(* PLC project TranslationStaging.project, CODESYS CODESYS V3.5 SP19 Patch 1 *)
(* stored: creationDateTime 2026-08-02T00:00:00, modificationDateTime 2026-08-02T00:00:00 *)

PROGRAM PRG_05_Translation_CFC
  VAR
    instTranslationArbiter : FB_TranslationArbiter;
    instSafetyTranslationM3 : FB_Safety_Translation;
    instTranslationRuntimeGate : FB_TranslationRuntimeGate;
    instTranslationM3 : FB_Translation;
    instTranslationFeedbackMemory : FB_TranslationFeedbackMemory;
    instTranslationRequestPublisher : FB_TranslationRequestPublisher;
    instTranslationCfcExpressions : FB_TranslationCfcExpressions;
  END_VAR
  VAR_OUTPUT
    TranslationFinalInterlockRequest : ST_TranslationFinalInterlockRequest;
    PowerCutOffRequested : BOOL;
    M3SafeStop : BOOL;
    M3PowerCutOff : BOOL;
    TranslationRequest : ST_TranslationFinalInterlockRequest;
  END_VAR

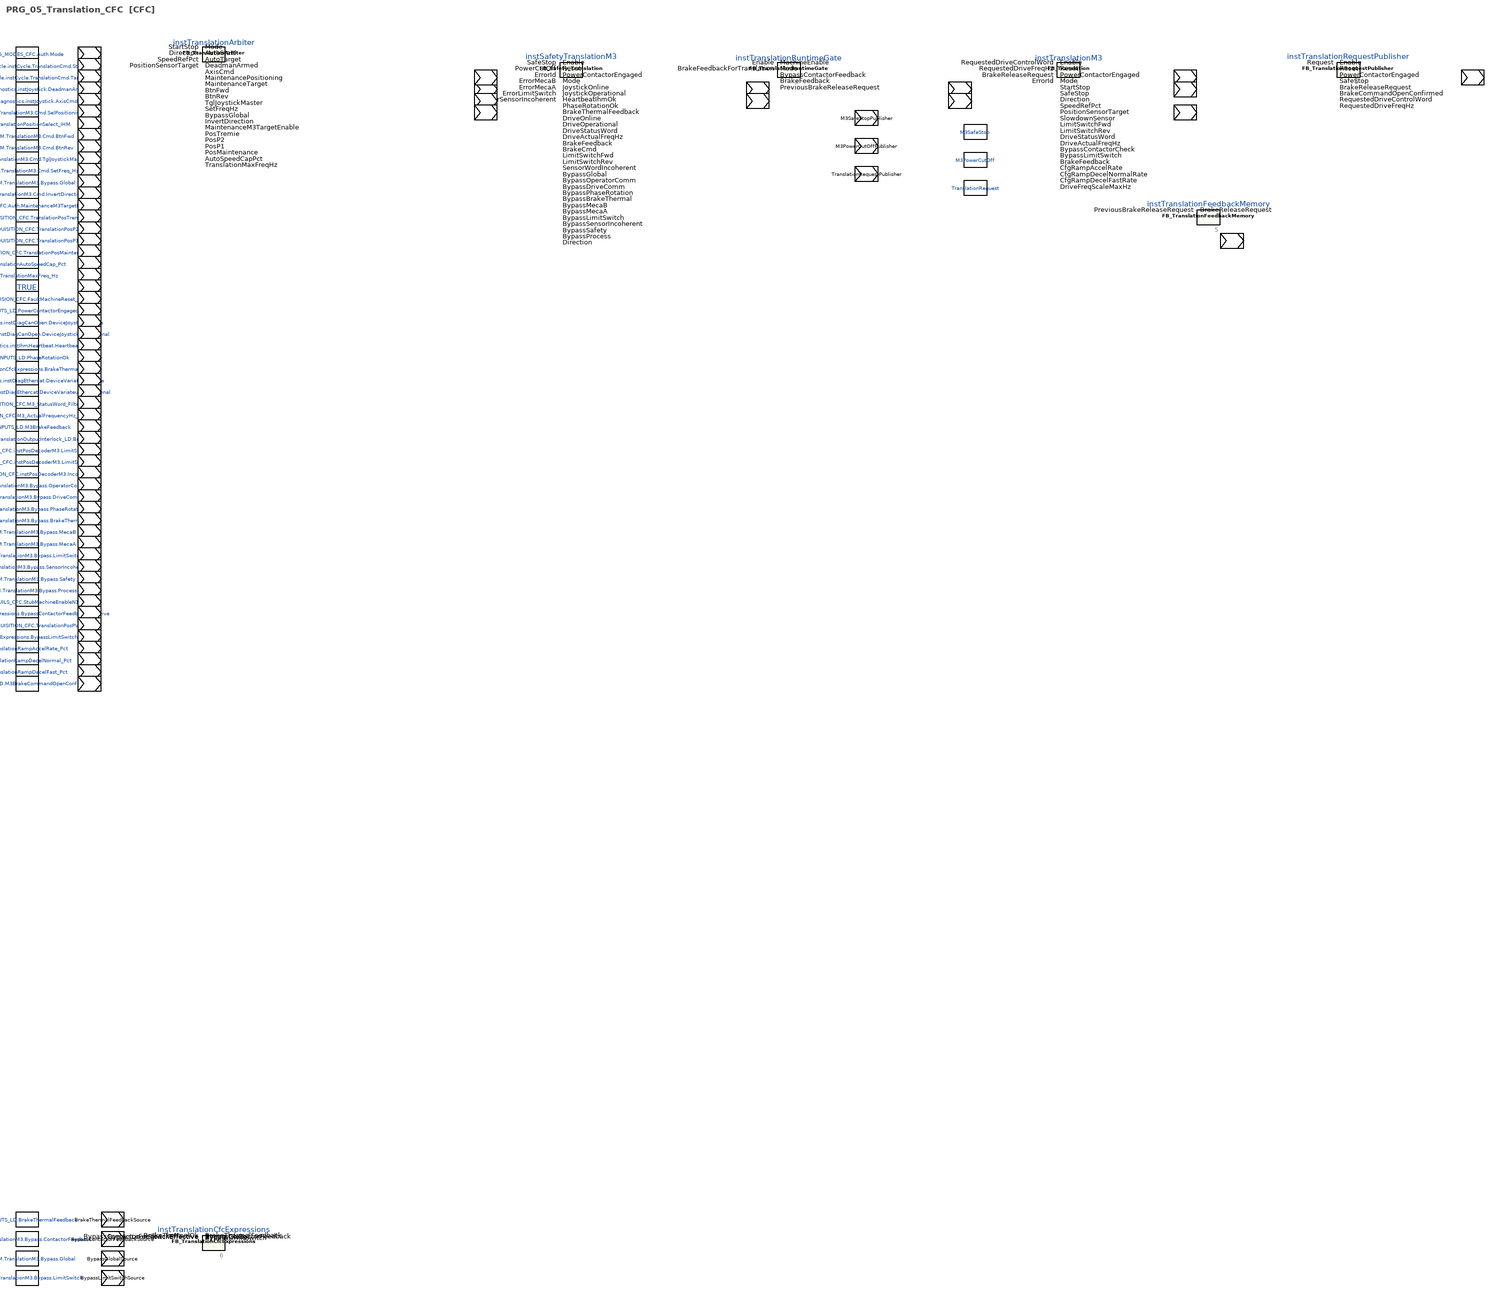
(* CFC diagram, written out as Structured Text *)
instTranslationArbiter(Mode := PRG_MODES_CFC.Auth.Mode, AutoStart := PRG_05_Cycle.instCycle.TranslationCmd.Start, AutoTarget := PRG_05_Cycle.instCycle.TranslationCmd.Target, DeadmanArmed := PRG_01_Diagnostics.instJoystick.DeadmanArmed, AxisCmd := PRG_01_Diagnostics.instJoystick.AxisCmdX, MaintenancePositioning := GVL_IHM.TranslationM3.Cmd.SelPositioning, MaintenanceTarget := StubTranslationPositionSelect_IHM, BtnFwd := GVL_IHM.TranslationM3.Cmd.BtnFwd, BtnRev := GVL_IHM.TranslationM3.Cmd.BtnRev, TglJoystickMaster := GVL_IHM.TranslationM3.Cmd.TglJoystickMaster, SetFreqHz := GVL_IHM.TranslationM3.Cmd.SetFreq_Hz, BypassGlobal := GVL_IHM.TranslationM3.Bypass.Global, InvertDirection := GVL_IHM.TranslationM3.Cmd.InvertDirection, MaintenanceM3TargetEnable := PRG_MODES_CFC.Auth.MaintenanceM3TargetEnable, PosTremie := PRG_ACQUISITION_CFC.TranslationPosTremie, PosP2 := PRG_ACQUISITION_CFC.TranslationPosP2, PosP1 := PRG_ACQUISITION_CFC.TranslationPosP1, PosMaintenance := PRG_ACQUISITION_CFC.TranslationPosMaintenance, AutoSpeedCapPct := _TranslationAutoSpeedCap_Pct, TranslationMaxFreqHz := _TranslationMaxFreq_Hz);
instSafetyTranslationM3(Enable := TRUE, Reset := PRG_SUPERVISION_CFC.FaultMachineReset_IHM, PowerContactorEngaged := PRG_INPUTS_LD.PowerContactorEngaged, Mode := PRG_MODES_CFC.Auth.Mode, JoystickOnline := PRG_01_Diagnostics.instDiagCanOpen.DeviceJoystick.Online, JoystickOperational := PRG_01_Diagnostics.instDiagCanOpen.DeviceJoystick.Operational, HeartbeatIhmOk := PRG_01_Diagnostics.instIhmHeartbeat.HeartbeatIhmOk, PhaseRotationOk := PRG_INPUTS_LD.PhaseRotationOk, BrakeThermalFeedback := instTranslationCfcExpressions.BrakeThermalOk, DriveOnline := PRG_01_Diagnostics.instDiagEthercat.DeviceVariateur.Online, DriveOperational := PRG_01_Diagnostics.instDiagEthercat.DeviceVariateur.Operational, DriveStatusWord := PRG_ACQUISITION_CFC.M3_StatusWord_Filtered, DriveActualFreqHz := PRG_ACQUISITION_CFC.M3_ActualFrequencyHz_Filtered, BrakeFeedback := PRG_INPUTS_LD.M3BrakeFeedback, BrakeCmd := GVL_Global.instTranslationOutputInterlock_LD.BrakeCmd, LimitSwitchFwd := PRG_ACQUISITION_CFC.instPosDecoderM3.LimitSwitchFwd, LimitSwitchRev := PRG_ACQUISITION_CFC.instPosDecoderM3.LimitSwitchRev, SensorWordIncoherent := PRG_ACQUISITION_CFC.instPosDecoderM3.Incoherent, BypassGlobal := GVL_IHM.TranslationM3.Bypass.Global, BypassOperatorComm := GVL_IHM.TranslationM3.Bypass.OperatorComm, BypassDriveComm := GVL_IHM.TranslationM3.Bypass.DriveComm, BypassPhaseRotation := GVL_IHM.TranslationM3.Bypass.PhaseRotation, BypassBrakeThermal := GVL_IHM.TranslationM3.Bypass.BrakeThermal, BypassMecaB := GVL_IHM.TranslationM3.Bypass.MecaB, BypassMecaA := GVL_IHM.TranslationM3.Bypass.MecaA, BypassLimitSwitch := GVL_IHM.TranslationM3.Bypass.LimitSwitch, BypassSensorIncoherent := GVL_IHM.TranslationM3.Bypass.SensorIncoherent, BypassSafety := GVL_IHM.TranslationM3.Bypass.Safety, BypassProcess := GVL_IHM.TranslationM3.Bypass.Process, Direction := instTranslationFeedbackMemory.PreviousBrakeReleaseRequest);
instTranslationRuntimeGate(MachineEnable := PRG_TREUILS_CFC.StubMachineEnableN1, Mode := PRG_MODES_CFC.Auth.Mode, BypassContactorFeedback := instTranslationCfcExpressions.BypassContactorFeedbackEffective, BrakeFeedback := PRG_INPUTS_LD.M3BrakeFeedback, PreviousBrakeReleaseRequest := instTranslationFeedbackMemory.PreviousBrakeReleaseRequest);
instTranslationM3(Enable := instTranslationFeedbackMemory.PreviousBrakeReleaseRequest, Reset := PRG_SUPERVISION_CFC.FaultMachineReset_IHM, PowerContactorEngaged := PRG_INPUTS_LD.PowerContactorEngaged, Mode := PRG_MODES_CFC.Auth.Mode, StartStop := instTranslationFeedbackMemory.PreviousBrakeReleaseRequest, SafeStop := instTranslationM3.RequestedDriveControlWord, Direction := instTranslationFeedbackMemory.PreviousBrakeReleaseRequest, SpeedRefPct := instTranslationFeedbackMemory.PreviousBrakeReleaseRequest, PositionSensorTarget := instTranslationRequestPublisher.Request, SlowdownSensor := PRG_ACQUISITION_CFC.TranslationPosPV, LimitSwitchFwd := PRG_ACQUISITION_CFC.instPosDecoderM3.LimitSwitchFwd, LimitSwitchRev := PRG_ACQUISITION_CFC.instPosDecoderM3.LimitSwitchRev, DriveStatusWord := PRG_ACQUISITION_CFC.M3_StatusWord_Filtered, DriveActualFreqHz := PRG_ACQUISITION_CFC.M3_ActualFrequencyHz_Filtered, BypassContactorCheck := GVL_IHM.TranslationM3.Bypass.Global, BypassLimitSwitch := instTranslationCfcExpressions.BypassLimitSwitchEffective, BrakeFeedback := instTranslationFeedbackMemory.PreviousBrakeReleaseRequest, CfgRampAccelRate := _TranslationRampAccelRate_Pct, CfgRampDecelNormalRate := _TranslationRampDecelNormal_Pct, CfgRampDecelFastRate := _TranslationRampDecelFast_Pct, DriveFreqScaleMaxHz := _TranslationMaxFreq_Hz);
instTranslationFeedbackMemory(BrakeReleaseRequest := instTranslationM3.BrakeReleaseRequest);
instTranslationRequestPublisher(Enable := PRG_TREUILS_CFC.StubMachineEnableN1, Reset := PRG_SUPERVISION_CFC.FaultMachineReset_IHM, PowerContactorEngaged := PRG_INPUTS_LD.PowerContactorEngaged, SafeStop := instTranslationM3.RequestedDriveControlWord, BrakeReleaseRequest := instTranslationM3.BrakeReleaseRequest, BrakeCommandOpenConfirmed := PRG_INPUTS_LD.M3BrakeCommandOpenConfirmed, RequestedDriveControlWord := instTranslationM3.RequestedDriveControlWord, RequestedDriveFreqHz := instTranslationM3.RequestedDriveFreqHz);
instTranslationCfcExpressions(BrakeThermalFeedback := PRG_INPUTS_LD.BrakeThermalFeedback, BypassContactorFeedback := GVL_IHM.TranslationM3.Bypass.ContactorFeedback, BypassGlobal := GVL_IHM.TranslationM3.Bypass.Global, BypassLimitSwitch := GVL_IHM.TranslationM3.Bypass.LimitSwitch);
M3SafeStop := instTranslationFeedbackMemory.PreviousBrakeReleaseRequest;
M3PowerCutOff := instTranslationFeedbackMemory.PreviousBrakeReleaseRequest;
TranslationRequest := instTranslationRequestPublisher.Request;
END_PROGRAM
